// TwinCAT 3 PLC project PLC_FrameworkOOP
// ProgramVersion: 3.1.4026.24
// CompilerDefines: VISU_USEPROPERTYINFO
// libraries:
//   Tc2_Standard, * (Beckhoff Automation GmbH)
//   Tc2_System, * (Beckhoff Automation GmbH)
// project tree:
//   Base/ Base.TcPOU
//   Devices/ I_DigitalInput.TcIO, DigitalInputNC.TcPOU, DigitalInputDummy.TcPOU, DigitalInputNO.TcPOU, DevicesExample.TcPOU, DevicesPolymorphismExample.TcPOU
//   ForceAbles/ Forceables.TcPOU, GVL_Forceables.TcGVL, ST_ForceAble.TcDUT
//   Forceable/ BoolSignal.TcPOU, BoolForceable.TcPOU, ForceableExample.TcPOU, I_Bool.TcIO, I_ForceableBOOL.TcIO
//   / GlobalTextList.TcGTLO, MAIN.TcPOU, PlcTask.TcTTO, Visualization Manager.TcVMO (not stored)
//   Logger/ GVL_Logger.TcGVL, I_Logger.TcIO, LoggerADS.TcPOU
// (motion and I/O tree: see PLC project plc_nooop)
// real-time tasks:
//   TASK PlcTask: cycle T#10ms, priority 20, ADS port 350
//   TASK PlcTask1: cycle T#10ms, priority 21, ADS port 351
//   TASK PlcTask2: cycle T#10ms, priority 22, ADS port 352

CONFIGURATION PLC_FrameworkOOP
    RESOURCE PLC ON TwinCAT3
        TASK PlcTask(INTERVAL := T#10ms, PRIORITY := 22);
        PROGRAM MAIN WITH PlcTask : MAIN;
    END_RESOURCE
END_CONFIGURATION

// ---- ForceAbles/ST_ForceAble.TcDUT
TYPE ST_ForceAble :
STRUCT
    name       : T_MaxString;
    path       : T_MaxString;
    value      : BOOL;
    forceValue : BOOL;
    forced     : BOOL;
END_STRUCT
END_TYPE

// ---- ForceAbles/GVL_Forceables.TcGVL
{attribute 'qualified_only'}
VAR_GLOBAL
    manager      : Forceables;
    arrForceables : ARRAY[0..MAXFORCEABLES - 1] OF ST_ForceAble;
END_VAR

VAR_GLOBAL CONSTANT
    MAXFORCEABLES : INT := 100;
END_VAR

// ---- Logger/GVL_Logger.TcGVL
{attribute 'qualified_only'}
VAR_GLOBAL
    logger          : LoggerADS;
END_VAR

// ---- Devices/I_DigitalInput.TcIO
INTERFACE I_DigitalInput

PROPERTY isActive : bool
GET
END_GET
END_PROPERTY

PROPERTY isNotActive : bool
GET
END_GET
END_PROPERTY

END_INTERFACE

// ---- Forceable/I_Bool.TcIO
INTERFACE I_Bool

PROPERTY value : BOOL
GET
END_GET
END_PROPERTY

END_INTERFACE

// ---- Forceable/I_ForceableBOOL.TcIO
INTERFACE I_ForceableBOOL EXTENDS I_Bool

PROPERTY name : STRING
GET
END_GET
END_PROPERTY

PROPERTY path : STRING
GET
END_GET
END_PROPERTY

METHOD force
VAR_INPUT
    forcedValue : BOOL;
END_VAR
END_METHOD

METHOD release
END_METHOD

PROPERTY isForced : BOOL
GET
END_GET
END_PROPERTY

END_INTERFACE

// ---- Logger/I_Logger.TcIO
INTERFACE I_Logger

METHOD trace
VAR_INPUT
	message						: T_MAXSTRING;  // STRING(255)
END_VAR
END_METHOD

END_INTERFACE

// ---- MAIN.TcPOU
PROGRAM MAIN

DevicesExample();
ForceableExample();
DevicesPolymorphismExample();
GVL_Forceables.manager.renew();

END_PROGRAM

// ---- Devices/DevicesExample.TcPOU
PROGRAM DevicesExample
VAR
    noInput         : DigitalInputNO('I201.1', GVL_Logger.logger);
    ncInput         : DigitalInputNC('I201.2', GVL_Logger.logger);
    dummyInput      : DigitalInputDummy('Undefined IO', GVL_Logger.logger);

    noActive        : BOOL;
    ncActive        : BOOL;
    dummyActive     : BOOL;

    noNotActive     : BOOL;
    ncNotActive     : BOOL;
    dummyNotActive  : BOOL;

    noName          : STRING;
    ncName          : STRING;
    dummyName       : STRING;

    noPath          : STRING;
    ncPath          : STRING;
    dummyPath       : STRING;

    traceAll        : BOOL;
    traceAllTrig    : R_TRIG;
END_VAR

noActive    := noInput.isActive;
ncActive    := ncInput.isActive;
dummyActive := dummyInput.isActive;

noNotActive    := noInput.isNotActive;
ncNotActive    := ncInput.isNotActive;
dummyNotActive := dummyInput.isNotActive;

noName    := noInput.name;
ncName    := ncInput.name;
dummyName := dummyInput.name;

noPath    := noInput.path;
ncPath    := ncInput.path;
dummyPath := dummyInput.path;

traceAllTrig(CLK := traceAll);
IF traceAllTrig.Q THEN
    noInput.trace(noInput.name);
    ncInput.trace(ncInput.name);
    dummyInput.trace(dummyInput.name);
END_IF

END_PROGRAM

// ---- Devices/DigitalInputNO.TcPOU
{attribute 'no_explicit_call' := 'DigitalInputNO is a class, do not call this POU directly, use a method'}
{attribute 'hide_all_locals'}
FUNCTION_BLOCK DigitalInputNO EXTENDS base IMPLEMENTS I_DigitalInput
VAR
    _input      AT %I*: BOOL;
END_VAR

PROPERTY isActive : bool
GET
isActive := _input;
END_GET
END_PROPERTY

PROPERTY isNotActive : bool
GET
isNotActive := NOT _input;
END_GET
END_PROPERTY

END_FUNCTION_BLOCK

// ---- Base/Base.TcPOU
{attribute 'no_explicit_call' := 'Base is a class, do not call this POU directly, use a method'}
{attribute 'hide_all_locals'}
{attribute 'reflection'}
FUNCTION_BLOCK ABSTRACT Base
VAR
    {attribute 'instance-path'}
    {attribute 'noinit'}
    _path   : T_MAXSTRING;

	// Locals 
   _name   : T_MAXSTRING;
    _logger : I_Logger;
END_VAR

METHOD FB_Init : BOOL
VAR_INPUT
    bInitRetains : BOOL;
    bInCopyCode  : BOOL;
    name         : STRING;
    logger       : I_Logger;
END_VAR
_name   := name;
_logger := logger;
END_METHOD

PROPERTY name : string
GET
name := _name;
END_GET
END_PROPERTY

PROPERTY path : string
GET
path := _path;
END_GET
END_PROPERTY

METHOD trace
VAR_INPUT
    message : T_MAXSTRING;
END_VAR
IF _logger <> 0 THEN
    _logger.trace(message);
ELSE
    ADSLOGSTR(msgCtrlMask := ADSLOG_MSGTYPE_HINT, msgFmtStr := message, strArg := '');
END_IF
END_METHOD

END_FUNCTION_BLOCK

// ---- Devices/DigitalInputNC.TcPOU
{attribute 'no_explicit_call' := 'DigitalInputNC is a class, do not call this POU directly, use a method'}
{attribute 'hide_all_locals'}
FUNCTION_BLOCK DigitalInputNC EXTENDS base IMPLEMENTS I_DigitalInput
VAR
    _input   AT %I* : BOOL;
    _signal  : BoolForceable(concat(name, ' forceable'), GVL_Logger.Logger);
END_VAR

METHOD FB_Init : BOOL
VAR_INPUT
    bInitRetains : BOOL;
    bInCopyCode  : BOOL;
    name         : STRING;
    logger       : I_Logger;
END_VAR
_signal.bind(_input);
END_METHOD

PROPERTY isActive : bool
GET
isActive := NOT _signal.value;
END_GET
END_PROPERTY

PROPERTY isNotActive : bool
GET
isNotActive := _signal.value;
END_GET
END_PROPERTY

PROPERTY signal : I_ForceableBOOL
GET
signal := _signal;
END_GET
END_PROPERTY

END_FUNCTION_BLOCK

// ---- Forceable/BoolForceable.TcPOU
{attribute 'no_explicit_call' := 'BoolForceable is a class, do not call this POU directly, use a method'}
{attribute 'hide_all_locals'}
FUNCTION_BLOCK BoolForceable EXTENDS BoolSignal IMPLEMENTS I_ForceableBOOL
VAR
    _forced   : BOOL;
    _isForced : BOOL;
END_VAR

METHOD FB_Init : BOOL
VAR_INPUT
    bInitRetains : BOOL;
    bInCopyCode  : BOOL;
    name         : STRING;
    logger       : I_Logger;
END_VAR
SUPER^.FB_Init(bInitRetains, bInCopyCode, name, logger);
IF name <> '' THEN
    GVL_Forceables.manager.register(THIS^);
END_IF
END_METHOD

METHOD force
VAR_INPUT
    forcedValue : BOOL;
END_VAR
_forced   := forcedValue;
_isForced := TRUE;
END_METHOD

METHOD release
_isForced := FALSE;
END_METHOD

PROPERTY value : BOOL
GET
IF _isForced THEN
    value := _forced;
ELSE
    value := SUPER^.value;
END_IF
END_GET
END_PROPERTY

PROPERTY isForced : BOOL
GET
isForced := _isForced;
END_GET
END_PROPERTY

END_FUNCTION_BLOCK

// ---- Forceable/BoolSignal.TcPOU
{attribute 'no_explicit_call' := 'BoolSignal is a class, do not call this POU directly, use a method'}
{attribute 'hide_all_locals'}
FUNCTION_BLOCK BoolSignal EXTENDS BASE IMPLEMENTS I_Bool
VAR
    _real : REFERENCE TO BOOL;
END_VAR

METHOD bind
VAR_IN_OUT
    signal : BOOL;
END_VAR
_real REF= signal;
END_METHOD

PROPERTY value : BOOL
GET
IF __ISVALIDREF(_real) THEN
    value := _real;
END_IF
END_GET
END_PROPERTY

END_FUNCTION_BLOCK

// ---- Devices/DigitalInputDummy.TcPOU
{attribute 'no_explicit_call' := 'DigitalInputDummy is a class, do not call this POU directly, use a method'}
{attribute 'hide_all_locals'}
FUNCTION_BLOCK DigitalInputDummy EXTENDS base IMPLEMENTS I_DigitalInput

PROPERTY isActive : BOOL
GET
isActive := true;
END_GET
END_PROPERTY

PROPERTY isNotActive : BOOL
GET
isNotActive := true;
END_GET
END_PROPERTY

END_FUNCTION_BLOCK

// ---- Forceable/ForceableExample.TcPOU
PROGRAM ForceableExample
VAR
    logger          : LoggerADS;

    // NC input: hardware reads TRUE when inactive, FALSE when active
    input           : DigitalInputNC('Door sensor', logger);

    // observed values — updated every scan via the proxy
    isActive        : BOOL;
    isNotActive     : BOOL;
    isForced        : BOOL;
    rawSignalValue  : BOOL;

    // force controls — set from online view
    forceActive     : BOOL;
    forceInactive   : BOOL;
    releaseForce    : BOOL;

    forceActiveTrig   : R_TRIG;
    forceInactiveTrig : R_TRIG;
    releaseTrig       : R_TRIG;
END_VAR

// read proxied values every scan
isActive       := input.isActive;
isNotActive    := input.isNotActive;
isForced       := input.signal.isForced;
rawSignalValue := input.signal.value;

// force the raw NC signal to FALSE  →  isActive = NOT FALSE = TRUE
// simulates: door sensor is activated (contact opened on NC wiring)
forceActiveTrig(CLK := forceActive);
IF forceActiveTrig.Q THEN
    input.signal.force(FALSE);
END_IF

// force the raw NC signal to TRUE  →  isActive = NOT TRUE = FALSE
// simulates: door sensor is inactive (contact closed at rest on NC wiring)
forceInactiveTrig(CLK := forceInactive);
IF forceInactiveTrig.Q THEN
    input.signal.force(TRUE);
END_IF

// release the force — isActive resumes following the real hardware input
releaseTrig(CLK := releaseForce);
IF releaseTrig.Q THEN
    input.signal.release();
END_IF

END_PROGRAM

// ---- Logger/LoggerADS.TcPOU
FUNCTION_BLOCK LoggerADS IMPLEMENTS I_Logger

METHOD trace
VAR_INPUT
	message	: T_MAXSTRING;
END_VAR
 ADSLOGSTR(msgCtrlMask := ADSLOG_MSGTYPE_HINT, msgFmtStr := message, strArg := '');
END_METHOD

END_FUNCTION_BLOCK

// ---- Devices/DevicesPolymorphismExample.TcPOU
PROGRAM DevicesPolymorphismExample
VAR
    noInput    : DigitalInputNO('Poly.NO', GVL_Logger.logger);
    ncInput    : DigitalInputNC('Poly.NC', GVL_Logger.logger);
    dummyInput : DigitalInputDummy('Poly.Dummy', GVL_Logger.logger);

    inputs      : ARRAY[0..2] OF I_DigitalInput;
    active      : ARRAY[0..2] OF BOOL;
	allActive	: BOOL;

    i           : INT;
    initialized : BOOL;
END_VAR

IF NOT initialized THEN
    inputs[0] := noInput;
    inputs[1] := ncInput;
    inputs[2] := dummyInput;
    initialized := TRUE;
END_IF

allActive := TRUE;
FOR i := 0 TO 2 DO
    IF inputs[i] <> 0 THEN
        active[i] := inputs[i].isActive;
		allActive := allActive AND active[i]; 
    END_IF
END_FOR

END_PROGRAM

// ---- ForceAbles/Forceables.TcPOU
{attribute 'no_explicit_call' := 'Forceables is a class, do not call this POU directly, use a method'}
{attribute 'hide_all_locals'}
FUNCTION_BLOCK Forceables
VAR
    _objects : ARRAY[0..GVL_Forceables.MAXFORCEABLES - 1] OF I_ForceableBOOL;
    _count   : INT;
END_VAR

METHOD register
VAR_INPUT
    obj : I_ForceableBOOL;
END_VAR
VAR
    i : INT;
END_VAR
IF obj = 0 THEN
    RETURN;
END_IF

FOR i := 0 TO GVL_Forceables.MAXFORCEABLES - 1 DO
    IF _objects[i] = obj THEN
        GVL_Forceables.arrForceables[i].name := obj.name;
        GVL_Forceables.arrForceables[i].path := obj.path;
        RETURN;
    END_IF
    IF _objects[i] = 0 THEN
        _objects[i] := obj;
        GVL_Forceables.arrForceables[i].name := obj.name;
        GVL_Forceables.arrForceables[i].path := obj.path;
        GVL_Forceables.arrForceables[i].value := obj.value;
        _count := _count + 1;
        RETURN;
    END_IF
END_FOR
END_METHOD

METHOD renew
VAR
    i : INT;
END_VAR
FOR i := 0 TO GVL_Forceables.MAXFORCEABLES - 1 DO
    IF _objects[i] = 0 THEN
        CONTINUE;
    END_IF
    IF GVL_Forceables.arrForceables[i].forced THEN
        _objects[i].force(GVL_Forceables.arrForceables[i].forceValue);
    ELSE
        _objects[i].release();
    END_IF
    GVL_Forceables.arrForceables[i].value := _objects[i].value;
END_FOR
END_METHOD

PROPERTY count : INT
GET
count := _count;
END_GET
END_PROPERTY

END_FUNCTION_BLOCK
